// TIA Portal project "SHE0024_Uloha_2" (V15.1)

(* hardware
DEVICE "S7-1200 station_1"  S7-1200 Station
   slot 0: "Rack_0"  S7-1200 Rack  Rack  V1.0
   slot 1: "PLC_1200_STUL_6"  CPU 1215C DC/DC/DC  6ES7 215-1AG40-0XB0  V4.3
DEVICE "ET 200S station_1"  ET 200S station
   slot 0: "Rack_0"  Rail
   slot 0: "et-stul-2"  IM 151-3 PN HF  6ES7 151-3BA23-0AB0  V7.0
   slot 1: "PM-E 24 to 48VDC_1"  PM-E 24 to 48VDC  6ES7 138-4CA50-0AB0
   slot 2: "2DI x 24VDC HF_1"  2DI x 24VDC HF  6ES7 131-4BB01-0AB0
   slot 3: "2DI x 24VDC HF_2"  2DI x 24VDC HF  6ES7 131-4BB01-0AB0
   slot 4: "2DI x 24VDC HF_3"  2DI x 24VDC HF  6ES7 131-4BB01-0AB0
   slot 5: "2DI x 24VDC HF_4"  2DI x 24VDC HF  6ES7 131-4BB01-0AB0
   slot 6: "2DI x 24VDC HF_5"  2DI x 24VDC HF  6ES7 131-4BB01-0AB0
   slot 7: "2DI x 24VDC HF_6"  2DI x 24VDC HF  6ES7 131-4BB01-0AB0
   slot 8: "2DI x 24VDC HF_7"  2DI x 24VDC HF  6ES7 131-4BB01-0AB0
   slot 9: "2DO x 24VDC / 0.5A HF_1"  2DO x 24VDC / 0.5A HF  6ES7 132-4BB01-0AB0
   slot 10: "2DO x 24VDC / 0.5A HF_2"  2DO x 24VDC / 0.5A HF  6ES7 132-4BB01-0AB0
   slot 11: "2DO x 24VDC / 0.5A HF_3"  2DO x 24VDC / 0.5A HF  6ES7 132-4BB01-0AB0
   slot 12: "2DO x 24VDC / 0.5A HF_4"  2DO x 24VDC / 0.5A HF  6ES7 132-4BB01-0AB0
   slot 13: "2AI x U ST_1"  2AI x U ST  6ES7 134-4FB01-0AB0
DEVICE "hmi-kpt700-stul-6"  KTP700 Basic PN
   slot 0: "hmi-kpt700-stul-6"  KTP700 Basic PN  6AV2 123-2GB03-0AX0  15.1.0.0
   slot 1: "HMI_RT_1"  KTP700 Basic PN  6AV2 123-2GB03-0AX0  15.1.0.0
   slot 5: "hmi-kpt700-stul-6.IE_CP_1"  PROFINET Interface  15.0.1.0
      slot 1: "PROFINET Interface_1"  PROFINET Interface
         slot 1: "Port_1"  Port
*)

// ===== PLC "PLC_1200_STUL_6"  CPU 1215C DC/DC/DC =====

VAR_GLOBAL   // PLC tag table "Default tag table"
   "ahjdkasd" AT %M5.0 : Bool;
   "START" AT %M0.0 : Bool;
   "cerv" AT %M0.1 : Bool;
   "modr" AT %M0.2 : Bool;
   "hlin" AT %M0.3 : Bool;
   "Nedef" AT %M0.4 : Bool;
   "magnet" AT %M0.5 : Bool;
   "tag1" AT %M0.6 : Bool;
   "tag2" AT %M0.7 : Bool;
   "tag3" AT %M1.0 : Bool;
   "Vyh_cerv" AT %M1.1 : Bool;
   "Vyh_modr" AT %M1.2 : Bool;
   "Vyh_hlin" AT %M1.3 : Bool;
   "Vyh_magnet" AT %M1.4 : Bool;
   "Tag_1" AT %MW250 : Int;
   "vyska" AT %MD6 : Real;
   "dira" AT %MD10 : Real;
   "STOP" AT %M1.5 : Bool;
   "pocet_modr" AT %MW2 : Int;
   "pocet_hlin" AT %MW14 : Int;
   "pocet_cerv_1" AT %MW16 : Int;
   "Reset_poctu" AT %M1.6 : Bool;
   "reset_modr" AT %M1.7 : Bool;
   "reset_hlin" AT %M4.0 : Bool;
   "reset_cerv_1" AT %M4.1 : Bool;
   "RCerv" AT %M4.2 : Bool;
   "Rhlin" AT %M4.3 : Bool;
   "RModr" AT %M4.4 : Bool;
END_VAR

VAR_GLOBAL   // PLC tag table "Tag table_1"
   "B1" AT %I72.0 : Bool;   // inkr snimac pas1
   "B2" AT %I72.1 : Bool;   // inkr snimac pas2
   "B3 Q1" AT %I73.0 : Bool;   // senzor cerv
   "B3 Q2" AT %I73.1 : Bool;   // senzor modr
   "B3 Q3" AT %I74.0 : Bool;   // senzor hlin
   "B3 Q4" AT %I74.1 : Bool;   // senzor nedef
   "B4" AT %I75.0 : Bool;   // snimac magn vlast
   "B6" AT %I75.1 : Bool;   // Snimac pritomnosti
   "B7" AT %I76.0 : Bool;   // zavora 1 z
   "B8" AT %I76.1 : Bool;   // zavora 1 v
   "B9" AT %I77.0 : Bool;   // vyrazec z
   "B10" AT %I77.1 : Bool;   // vyrazec v
   "B11" AT %I78.0 : Bool;   // zavora 2 z
   "B12" AT %I78.1 : Bool;   // zavora 2 v
   "Y 1" AT %Q69.0 : Bool;   // zavora1
   "Y 2" AT %Q69.1 : Bool;   // vyrazec
   "Y 3" AT %Q70.0 : Bool;   // zavora2
   "Y 4" AT %Q70.1 : Bool;   // aktivace - snimac vysky
   "Y M1" AT %Q71.0 : Bool;   // pas 1
   "Y M2" AT %Q71.1 : Bool;   // pas 2
   "B5" AT %IW68 : Word;   // senzor vysky
END_VAR

VAR_GLOBAL CONSTANT   // PLC tag table "Tag table_1"
   "zacatek_cyklu" : Int := 0;
   "detekce_barev" : Int := 2;
   "snimani_magnet" : Int := 3;
   "aktivace_zavory1" : Int := 4;
   "deaktivace_zavory1" : Int := 5;
   "aktivace_zavory2" : Int := 6;
   "aktivace vyrazecu" : Int := 7;
   "deaktivace vyrazecu" : Int := 8;
   "reset_cerv" : Int := 0;
END_VAR

VAR_GLOBAL   // PLC tag table "Tag table_2"
   "Cyklus" AT %MW20 : Int;
   "Count" AT %MW22 : Int;
END_VAR

VAR_GLOBAL   // PLC tag table "Tag table_3"
   "TestBool" AT %M400.0 : Bool;
   "TestInt" AT %MW401 : Int;
   "TestReal" AT %MD404 : Real;
END_VAR

DATA_BLOCK "Block_1_DB"   // DB4
{ S7_Optimized_Access := 'TRUE' }
VERSION : 0.1
// stored: InstanceOfName Block_1
"Block_1"
BEGIN
END_DATA_BLOCK

// folder: System blocks/Program resources

DATA_BLOCK "IEC_Timer_0_DB"   // DB1
{ S7_Optimized_Access := 'TRUE' }
AUTHOR : Simatic
FAMILY : IEC
NAME : IEC_TMR
VERSION : 1.0
// stored: InstanceOfName IEC_TIMER
"IEC_TIMER"
BEGIN
END_DATA_BLOCK

DATA_BLOCK "IEC_Timer_0_DB_1"   // DB2
{ S7_Optimized_Access := 'TRUE' }
AUTHOR : Simatic
FAMILY : IEC
NAME : IEC_TMR
VERSION : 1.0
// stored: InstanceOfName IEC_TIMER
"IEC_TIMER"
BEGIN
END_DATA_BLOCK

DATA_BLOCK "IEC_Timer_0_DB_2"   // DB3
{ S7_Optimized_Access := 'TRUE' }
AUTHOR : Simatic
FAMILY : IEC
NAME : IEC_TMR
VERSION : 1.0
// stored: InstanceOfName IEC_TIMER
"IEC_TIMER"
BEGIN
END_DATA_BLOCK

DATA_BLOCK "IEC_Timer_0_DB_3"   // DB5
{ S7_Optimized_Access := 'TRUE' }
AUTHOR : Simatic
FAMILY : IEC
NAME : IEC_TMR
VERSION : 1.0
// stored: InstanceOfName IEC_TIMER
"IEC_TIMER"
BEGIN
END_DATA_BLOCK

DATA_BLOCK "IEC_Timer_0_DB_4"   // DB6
{ S7_Optimized_Access := 'TRUE' }
AUTHOR : Simatic
FAMILY : IEC
NAME : IEC_TMR
VERSION : 1.0
// stored: InstanceOfName IEC_TIMER
"IEC_TIMER"
BEGIN
END_DATA_BLOCK

DATA_BLOCK "IEC_Timer_0_DB_5"   // DB7
{ S7_Optimized_Access := 'TRUE' }
AUTHOR : Simatic
FAMILY : IEC
NAME : IEC_TMR
VERSION : 1.0
// stored: InstanceOfName IEC_TIMER
"IEC_TIMER"
BEGIN
END_DATA_BLOCK

DATA_BLOCK "IEC_Timer_0_DB_6"   // DB8
{ S7_Optimized_Access := 'TRUE' }
AUTHOR : Simatic
FAMILY : IEC
NAME : IEC_TMR
VERSION : 1.0
// stored: InstanceOfName IEC_TIMER
"IEC_TIMER"
BEGIN
END_DATA_BLOCK

DATA_BLOCK "IEC_Counter_0_DB"   // DB9
{ S7_Optimized_Access := 'TRUE' }
AUTHOR : Simatic
FAMILY : IEC
NAME : CNTR
VERSION : 1.0
// stored: InstanceOfName IEC_COUNTER
"IEC_COUNTER"
BEGIN
END_DATA_BLOCK

DATA_BLOCK "IEC_Timer_0_DB_8"   // DB10
{ S7_Optimized_Access := 'TRUE' }
AUTHOR : Simatic
FAMILY : IEC
NAME : IEC_TMR
VERSION : 1.0
// stored: InstanceOfName IEC_TIMER
"IEC_TIMER"
BEGIN
END_DATA_BLOCK

DATA_BLOCK "IEC_Counter_0_DB_1"   // DB11
{ S7_Optimized_Access := 'TRUE' }
AUTHOR : Simatic
FAMILY : IEC
NAME : CNTR
VERSION : 1.0
// stored: InstanceOfName IEC_COUNTER
"IEC_COUNTER"
BEGIN
END_DATA_BLOCK

DATA_BLOCK "IEC_Counter_0_DB_2"   // DB12
{ S7_Optimized_Access := 'TRUE' }
AUTHOR : Simatic
FAMILY : IEC
NAME : CNTR
VERSION : 1.0
// stored: InstanceOfName IEC_COUNTER
"IEC_COUNTER"
BEGIN
END_DATA_BLOCK

// folder: (top level)

FUNCTION_BLOCK "Block_1"   // FB1, LAD
{ S7_Optimized_Access := 'TRUE' }
VERSION : 0.1
   VAR_TEMP   // added for the SCL form of the ladder/FBD networks
      _w1 : Bool;
      _w2 : Bool;
      _w3 : Bool;
      _w4 : Bool;
   END_VAR
BEGIN

REGION Network 1: Aktivace - zacatek cyklu
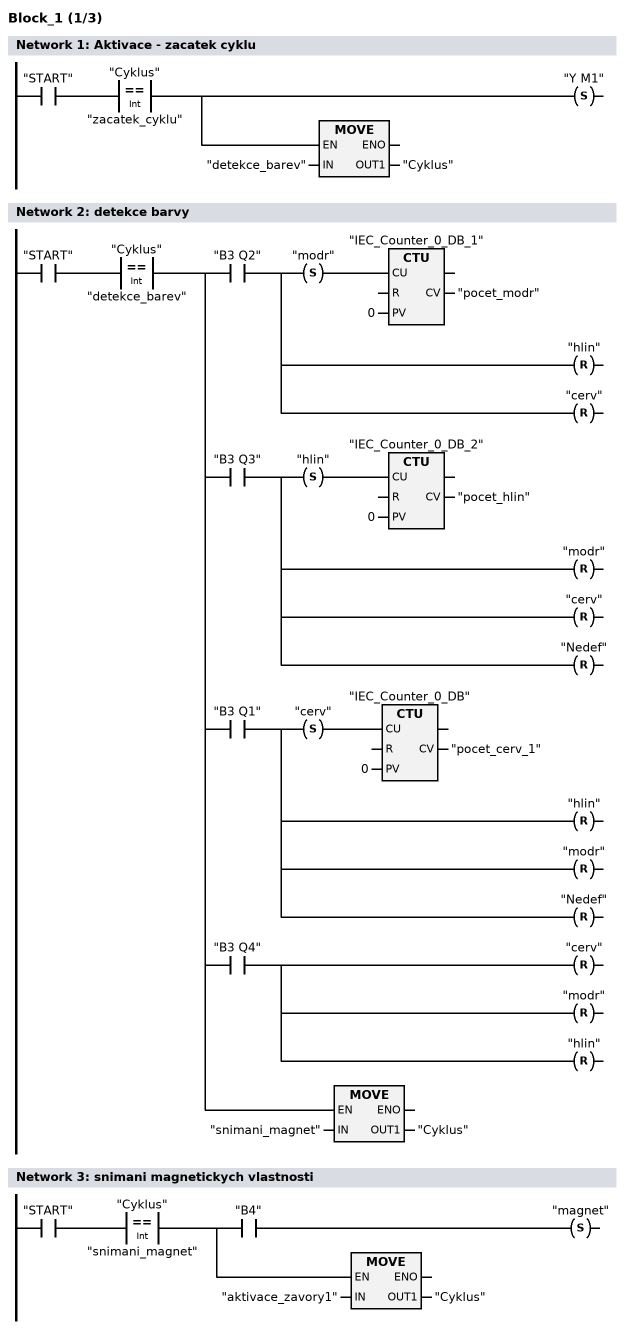
   RUNG wire#powerrail
      Contact( "START" )
      { S7_Templates := "SrcType := Int" } EQ_Contact(in1 := "Cyklus", in2 := "zacatek_cyklu")
      wire#w1
      S_Coil( "Y M1" )
   END_RUNG
   RUNG wire#w1
      Move(in := "detekce_barev", out1 => "Cyklus")
   END_RUNG
   // the same network as SCL:
   IF "START" AND ("Cyklus" = "zacatek_cyklu") THEN
       "Y M1" := TRUE;
       "Cyklus" := "detekce_barev";
   END_IF;
END_REGION

REGION Network 2: detekce barvy
   #_w1 := "START" AND ("Cyklus" = "detekce_barev");
   #_w2 := #_w1 AND "B3 Q2";
   IF #_w2 THEN "modr" := TRUE; END_IF;
   "IEC_Counter_0_DB_1".CTU(CU := #_w2, PV := 0, CV => "pocet_modr");
   IF #_w2 THEN
       "hlin" := FALSE;
       "cerv" := FALSE;
   END_IF;
   #_w3 := #_w1 AND "B3 Q3";
   IF #_w3 THEN "hlin" := TRUE; END_IF;
   "IEC_Counter_0_DB_2".CTU(CU := #_w3, PV := 0, CV => "pocet_hlin");
   IF #_w3 THEN
       "modr" := FALSE;
       "cerv" := FALSE;
       "Nedef" := FALSE;
   END_IF;
   #_w4 := #_w1 AND "B3 Q1";
   IF #_w4 THEN "cerv" := TRUE; END_IF;
   "IEC_Counter_0_DB".CTU(CU := #_w4, PV := 0, CV => "pocet_cerv_1");
   IF #_w4 THEN
       "hlin" := FALSE;
       "modr" := FALSE;
       "Nedef" := FALSE;
   END_IF;
   IF #_w1 AND "B3 Q4" THEN
       "cerv" := FALSE;
       "modr" := FALSE;
       "hlin" := FALSE;
   END_IF;
   IF #_w1 THEN "Cyklus" := "snimani_magnet"; END_IF;
END_REGION

REGION Network 3: snimani magnetickych vlastnosti
   RUNG wire#powerrail
      Contact( "START" )
      { S7_Templates := "SrcType := Int" } EQ_Contact(in1 := "Cyklus", in2 := "snimani_magnet")
      wire#w1
      Contact( "B4" )
      S_Coil( "magnet" )
   END_RUNG
   RUNG wire#w1
      Move(in := "aktivace_zavory1", out1 => "Cyklus")
   END_RUNG
   // the same network as SCL:
   #_w1 := "START" AND ("Cyklus" = "snimani_magnet");
   IF #_w1 AND "B4" THEN "magnet" := TRUE; END_IF;
   IF #_w1 THEN "Cyklus" := "aktivace_zavory1"; END_IF;
END_REGION

REGION Network 4: aktivace zavory 1
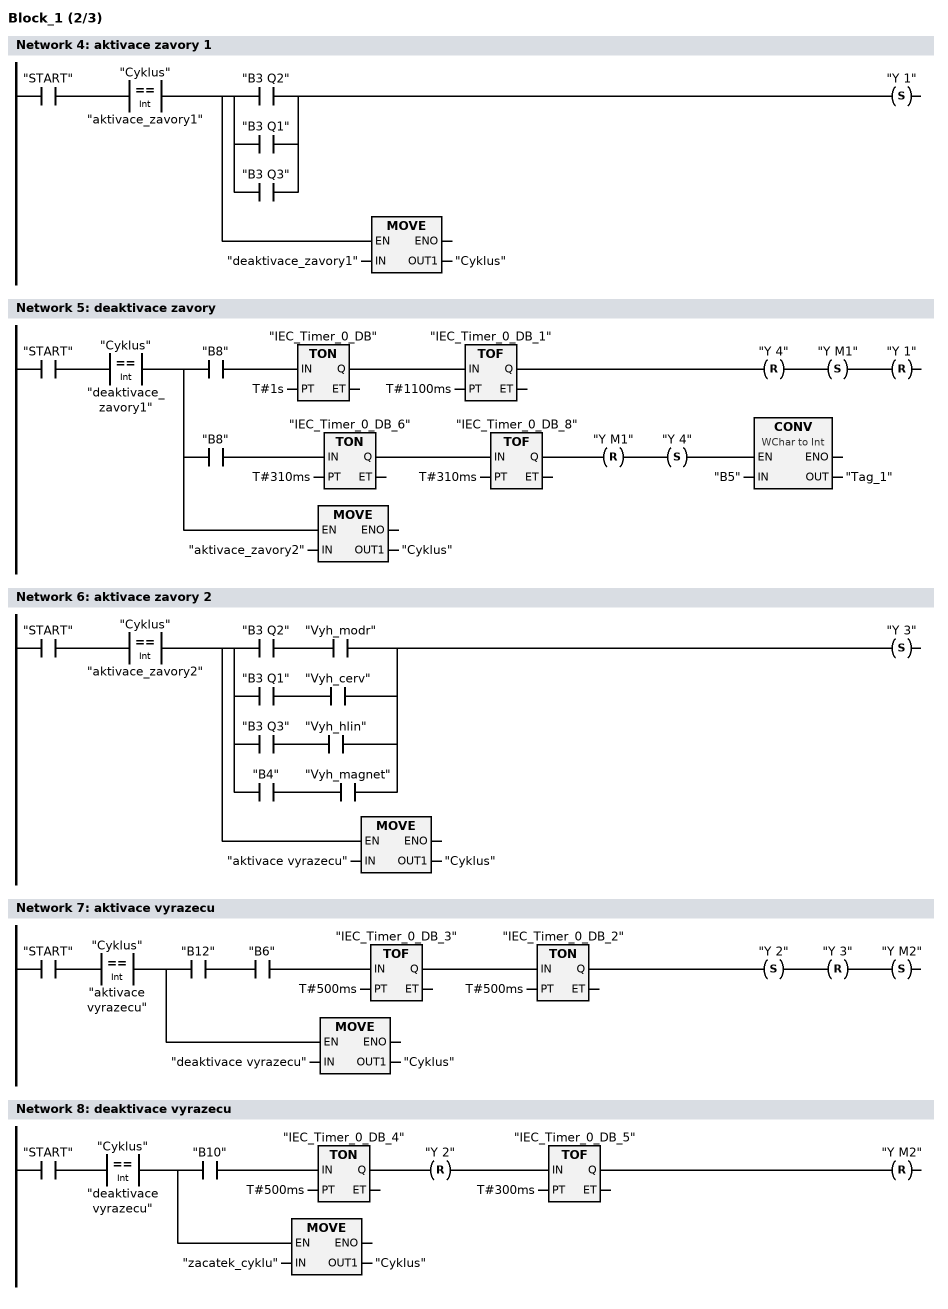
   RUNG wire#powerrail
      Contact( "START" )
      { S7_Templates := "SrcType := Int" } EQ_Contact(in1 := "Cyklus", in2 := "aktivace_zavory1")
      wire#w1
      Contact( "B3 Q2" )
      wire#w2
      S_Coil( "Y 1" )
   END_RUNG
   RUNG wire#w1
      Contact( "B3 Q1" )
   END_RUNG wire#w2
   RUNG wire#w1
      Contact( "B3 Q3" )
   END_RUNG wire#w2
   RUNG wire#w1
      Move(in := "deaktivace_zavory1", out1 => "Cyklus")
   END_RUNG
   // the same network as SCL:
   #_w1 := "START" AND ("Cyklus" = "aktivace_zavory1");
   IF #_w1 AND ("B3 Q2" OR "B3 Q1" OR "B3 Q3") THEN "Y 1" := TRUE; END_IF;
   IF #_w1 THEN "Cyklus" := "deaktivace_zavory1"; END_IF;
END_REGION

REGION Network 5: deaktivace zavory
   #_w1 := "START" AND ("Cyklus" = "deaktivace_zavory1");
   "IEC_Timer_0_DB".TON(IN := #_w1 AND "B8", PT := T#1s);
   "IEC_Timer_0_DB_1".TOF(IN := "IEC_Timer_0_DB".Q, PT := T#1100ms);
   IF "IEC_Timer_0_DB_1".Q THEN
       "Y 4" := FALSE;
       "Y M1" := TRUE;
       "Y 1" := FALSE;
   END_IF;
   "IEC_Timer_0_DB_6".TON(IN := #_w1 AND "B8", PT := T#310ms);
   "IEC_Timer_0_DB_8".TOF(IN := "IEC_Timer_0_DB_6".Q, PT := T#310ms);
   IF "IEC_Timer_0_DB_8".Q THEN
       "Y M1" := FALSE;
       "Y 4" := TRUE;
       "Tag_1" := WCHAR_TO_INT("B5");
   END_IF;
   IF #_w1 THEN "Cyklus" := "aktivace_zavory2"; END_IF;
END_REGION

REGION Network 6: aktivace zavory 2
   RUNG wire#powerrail
      Contact( "START" )
      { S7_Templates := "SrcType := Int" } EQ_Contact(in1 := "Cyklus", in2 := "aktivace_zavory2")
      wire#w1
      Contact( "B3 Q2" )
      Contact( "Vyh_modr" )
      wire#w2
      S_Coil( "Y 3" )
   END_RUNG
   RUNG wire#w1
      Contact( "B3 Q1" )
      Contact( "Vyh_cerv" )
   END_RUNG wire#w2
   RUNG wire#w1
      Contact( "B3 Q3" )
      Contact( "Vyh_hlin" )
   END_RUNG wire#w2
   RUNG wire#w1
      Contact( "B4" )
      Contact( "Vyh_magnet" )
   END_RUNG wire#w2
   RUNG wire#w1
      Move(in := "aktivace vyrazecu", out1 => "Cyklus")
   END_RUNG
   // the same network as SCL:
   #_w1 := "START" AND ("Cyklus" = "aktivace_zavory2");
   IF #_w1 AND (("B3 Q2" AND "Vyh_modr") OR ("B3 Q1" AND "Vyh_cerv") OR ("B3 Q3" AND "Vyh_hlin") OR ("B4" AND "Vyh_magnet")) THEN
       "Y 3" := TRUE;
   END_IF;
   IF #_w1 THEN "Cyklus" := "aktivace vyrazecu"; END_IF;
END_REGION

REGION Network 7: aktivace vyrazecu
   #_w1 := "START" AND ("Cyklus" = "aktivace vyrazecu");
   "IEC_Timer_0_DB_3".TOF(IN := #_w1 AND "B12" AND "B6", PT := T#500ms);
   "IEC_Timer_0_DB_2".TON(IN := "IEC_Timer_0_DB_3".Q, PT := T#500ms);
   IF "IEC_Timer_0_DB_2".Q THEN
       "Y 2" := TRUE;
       "Y 3" := FALSE;
       "Y M2" := TRUE;
   END_IF;
   IF #_w1 THEN "Cyklus" := "deaktivace vyrazecu"; END_IF;
END_REGION

REGION Network 8: deaktivace vyrazecu
   #_w1 := "START" AND ("Cyklus" = "deaktivace vyrazecu");
   "IEC_Timer_0_DB_4".TON(IN := #_w1 AND "B10", PT := T#500ms);
   IF "IEC_Timer_0_DB_4".Q THEN "Y 2" := FALSE; END_IF;
   "IEC_Timer_0_DB_5".TOF(IN := "IEC_Timer_0_DB_4".Q, PT := T#300ms);
   IF "IEC_Timer_0_DB_5".Q THEN "Y M2" := FALSE; END_IF;
   IF #_w1 THEN "Cyklus" := "zacatek_cyklu"; END_IF;
END_REGION

REGION Network 9: zpracovani analagove hodnoty
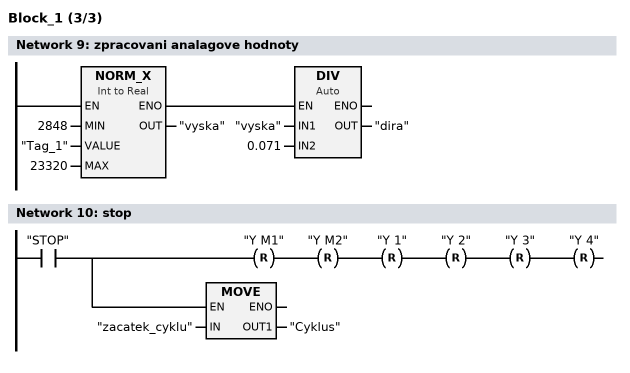
   RUNG wire#powerrail
      { S7_Templates := "[SrcType := Int, DestType := Real]" } Normalize(min := 2848, value := "Tag_1", max := 23320, out => "vyska")
      Div(in1 := "vyska", in2 := 0.071, out => "dira")
   END_RUNG
   // the same network as SCL:
   "vyska" := NORM_X(MIN := 2848, VALUE := "Tag_1", MAX := 23320);
   "dira" := "vyska" / 0.071;
END_REGION

REGION Network 10: stop
   RUNG wire#powerrail
      Contact( "STOP" )
      wire#w1
      R_Coil( "Y M1" )
      R_Coil( "Y M2" )
      R_Coil( "Y 1" )
      R_Coil( "Y 2" )
      R_Coil( "Y 3" )
      R_Coil( "Y 4" )
   END_RUNG
   RUNG wire#w1
      Move(in := "zacatek_cyklu", out1 => "Cyklus")
   END_RUNG
   // the same network as SCL:
   IF "STOP" THEN
       "Y M1" := FALSE;
       "Y M2" := FALSE;
       "Y 1" := FALSE;
       "Y 2" := FALSE;
       "Y 3" := FALSE;
       "Y 4" := FALSE;
       "Cyklus" := "zacatek_cyklu";
   END_IF;
END_REGION
END_FUNCTION_BLOCK

ORGANIZATION_BLOCK "Main"   // OB1, FBD, ProgramCycle
TITLE = "Main Program Sweep (Cycle)"
{ S7_Optimized_Access := 'TRUE' }
VERSION : 0.1
   VAR_INPUT
      Initial_Call : Bool;   // Initial call of this OB
      Remanence : Bool;   // =True, if remanent data are available
   END_VAR
BEGIN

REGION Network 1
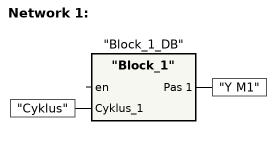
   "Block_1_DB"(Cyklus_1 := "Cyklus", "Pas 1" => "Y M1");   // "Block_1"
END_REGION
END_ORGANIZATION_BLOCK

(* ===== HMI "HMI_RT_1" =====
system functions are stored by id; their names below are inferred from use
connection "HMI_Connection_1": ETHERNET, SMART_S7_1200_OMS

HMI tags "Default tag table"
   "Tag_ScreenNumber" : UInt, internal
   "TestBool" : Bool = PLC TestBool AT %M400.0, 1 s
   "TestInt" : Int = PLC TestInt AT %MW401, 1 s
   "TestReal" : Real = PLC TestReal AT %MD404, 1 s
   "START" : Bool = PLC START AT %M0.0, 1 s
   "STOP" : Bool = PLC STOP AT %M1.5, 1 s
   "pocet_modr" : Int = PLC pocet_modr AT %MW2, 1 s
   "pocet_hlin" : Int = PLC pocet_hlin AT %MW14, 1 s
   "dira" : Real = PLC dira AT %MD10, 1 s
   "Vyh_cerv" : Bool = PLC Vyh_cerv AT %M1.1, 1 s
   "modr" : Bool = PLC modr AT %M0.2, 1 s
   "hlin" : Bool = PLC hlin AT %M0.3, 1 s
   "Vyh_magnet" : Bool = PLC Vyh_magnet AT %M1.4, 1 s
   "Vyh_hlin" : Bool = PLC Vyh_hlin AT %M1.3, 1 s
   "Vyh_modr" : Bool = PLC Vyh_modr AT %M1.2, 1 s
   "pocet_cerv_1" : Int = PLC pocet_cerv_1 AT %MW16, 1 s
   "cerv" : Bool = PLC cerv AT %M0.1, 1 s
   "reset_modr" : Bool = PLC reset_modr AT %M1.7, 1 s
   "reset_hlin" : Bool = PLC reset_hlin AT %M4.0, 1 s
   "reset_cerv_1" : Bool = PLC reset_cerv_1 AT %M4.1, 1 s

analog alarms
   1: 'varovani', class Errors, trigger "pocet_hlin"

Template "Template_1" 800x480
   Button "Alarms" at 1,52 size 71x50; TextOff 'Alarms'; PictureOff "AlarmDisplay_KTP700_Basic_PN_TR"; PictureOn "AlarmDisplay_KTP700_Basic_PN_TR"
      on Release: function_ef3f5d25("Alarm window_Unacknowledged", -1)
   Button "Start screen" at 1,106 size 71x50; TextOff 'Start screen'; PictureOff "NavigateHome_KTP700_Basic_PN_TR"; PictureOn "NavigateHome_KTP700_Basic_PN_TR"
      on Release: ActivateScreen("Main", 0)
      on Click: ActivateScreen("Main", 0)
   Button "Log on" at 1,159 size 71x50; TextOff 'Log on'; PictureOff "Login_KTP700_Basic_PN_TR"; PictureOn "Login_KTP700_Basic_PN_TR"
      on Release: function_a2a04561()
      on Click: function_a2a04561()
   Button "Template_Button" at 1,213 size 71x50; TextOff 'Text'
   Button "Template_Button_1" at 1,267 size 71x50; TextOff 'Text'
   Button "Template_Button_2" at 1,321 size 71x50; TextOff 'Text'
   Button "Template_Button_3" at 1,374 size 71x50; TextOff 'Text'
   Button "Exit" at 1,428 size 71x50; TextOff 'Exit'; PictureOff "ExitRuntime_KTP700_Basic_PN_TR"; PictureOn "ExitRuntime_KTP700_Basic_PN_TR"
      on Release: StopRuntime(0)
   SymbolicIOField "Symbolic_IO_Field_Screen" at 93,9 size 600x33; TextOff '0'; TextOn '1'; TextList "TextList_ScreenNames"
      ProcessValue <- "Tag_ScreenNumber"
      on Change: ActivateScreenByNumber("Tag_ScreenNumber", 0)
   DateTimeField "HmiScreenItemData" at 695,25 size 105x25
   DateTimeField "HmiScreenItemData_1" at 695,0 size 105x25
   GraphicView "Logo" at 0,0 size 91x51; Picture "Logo of hmi-kpt700-stul-7"

screen "Main" 800x480, template "Template_1"
   on GenerateScreen: SetTag("Tag_ScreenNumber", 1)
   TextField "HmiScreenItemData" at 105,43 size 582x25; Text 'Pracoviště testovací'
   IOField "I/O field_1" at 106,161 size 96x32; FormatPattern 999
      ProcessValue <- "pocet_modr"
   Button "Button_1" at 109,90 size 96x32; TextOff 'START'
      Appearance <- "START"
      on Press: SetBit("START"); ResetBit("STOP")
   Button "Button_2" at 584,88 size 96x32; TextOff 'STOP'
      Appearance <- "STOP"
      on Press: SetBit("STOP"); ResetBit("START")
   Circle "Circle_1" at 382,90 size 34x34
      Appearance <- "START"
   IOField "I/O field_2" at 105,234 size 96x32; FormatPattern 999
      ProcessValue <- "pocet_hlin"
   TextField "HmiScreenItemData_1" at 0,195 size 582x25; Text 'Text'
   TextField "Text field_1" at 109,202 size 192x23; Text 'Pocet hliníkových puků'
   TextField "Text field_2" at 101,120 size 170x23; Text 'Pocet modrých puků'
   TextField "Text field_3" at 111,340 size 39x23; Text 'Díra'
   IOField "I/O field_3" at 109,364 size 96x32; FormatPattern 99.999
      ProcessValue <- "dira"
   TextField "Text field_4" at 205,366 size 35x23; Text 'mm'
   TextField "Text field_5" at 201,243 size 33x23; Text 'kus'
   TextField "Text field_6" at 207,170 size 33x23; Text 'kus'
   Button "Button_4" at 292,408 size 96x32; TextOff 'Graf'
      on Activate: ActivateScreen("Trend", 2)
   Button "Button_5" at 101,408 size 157x32; TextOff 'Změna parametru'; Authorization "Operate"
      on Click: ActivateScreen("Parametrs", 0)
   TextField "Text field_7" at 101,276 size 182x23; Text 'Pocet červených puků'
   IOField "I/O field_4" at 106,301 size 96x32; FormatPattern 999
      ProcessValue <- "pocet_cerv_1"
   TextField "Text field_8" at 202,310 size 33x23; Text 'kus'
   GraphicView "Graphic view_1" at 699,378 size 101x102; Picture "fei"

screen "Parametrs" 800x480
   Button "Button_1" at 316,18 size 171x31; TextOff 'Vrátit se na hlavní'
      on Click: ActivateScreen("Main", 0)
   Button "Button_2" at 19,105 size 171x31; TextOff 'Vyřadit modré'
      on Click: SetBit("Vyh_modr")
   Button "Button_3" at 23,160 size 171x31; TextOff 'Vyřadit hliníkové'
      on Click: SetBit("Vyh_hlin")
   TextField "Text field_1" at 13,70 size 156x23; Text 'Vyřazeni dle barvy'
   TextField "Text field_2" at 19,273 size 307x23; Text 'Vyřazeni dle magnetických vlastností'
   Button "Button_4" at 19,310 size 171x31; TextOff 'Vyřadit magnety'
      on Click: SetBit("Vyh_magnet")
   Button "Button_6" at 214,105 size 171x31; TextOff 'Zrušit'
      on Click: ResetBit("Vyh_modr")
   Button "Button_7" at 214,160 size 171x31; TextOff 'Zrušit'
      on Click: ResetBit("Vyh_hlin")
   Button "Button_8" at 210,310 size 171x31; TextOff 'Zrušit'
      on Click: ResetBit("Vyh_hlin")
   Button "Button_5" at 23,212 size 171x31; TextOff 'Vyřadit červené'
      on Click: SetBit("Vyh_cerv")
   Button "Button_9" at 216,212 size 171x31; TextOff 'Zrušit'
      on Click: ResetBit("Vyh_cerv")

screen "Trend" 800x480
   Button "Button_1" at 323,23 size 182x32; TextOff 'Vrátit se na hlavní'
      on Activate: ActivateScreen("Main", 0)
   TrendView "Trend view_1" at 143,113 size 600x300
*)